FUNCTION_BLOCK "PIDControl"
{ S7_Optimized_Access := 'TRUE' }
VERSION : 0.1
AUTHOR : 'AI_Generated'

VAR_INPUT
    bEnable : Bool;                    // PID 使能
    bReset : Bool;                     // 积分复位
    bManualMode : Bool;                // 手动模式
    rSetpoint : Real;                  // 设定值 (工程单位)
    rProcessValue : Real;              // 过程值 (工程单位)
    rManualValue : Real;               // 手动输出值 (%)
    rKp : Real;                        // 比例增益
    rTi : Real;                        // 积分时间 (秒，0=无积分)
    rTd : Real;                        // 微分时间 (秒，0=无微分)
    rOutputMin : Real;                 // 输出下限 (%)
    rOutputMax : Real;                 // 输出上限 (%)
    rSetpointRampRate : Real;          // 设定值斜坡速率 (单位/秒)
    rDeadband : Real;                  // 死区 (工程单位)
END_VAR

VAR_OUTPUT
    rControlOutput : Real;             // 控制输出 (%)
    rError : Real;                     // 偏差值
    rP : Real;                         // P 分量
    rI : Real;                         // I 分量
    rD : Real;                         // D 分量
    bLimiting : Bool;                  // 输出限幅中
    bAntiWindupActive : Bool;          // 抗饱和激活
    bRampActive : Bool;                // 斜坡进行中
    rSetpointRamped : Real;            // 斜坡后的设定值
END_VAR

VAR
    // PID 内部变量
    rIntegral : Real;                  // 积分累加值
    rIntegralInc : Real;               // 本次积分增量（只计算一次）
    rPrevError : Real;                 // 上次偏差
    rPrevPV : Real;                    // 上次过程值（用于微分）
    rSampleTime : Real;                // 采样时间 (秒)
    rOutput : Real;                    // 计算输出

    // 设定值斜坡
    rRampTarget : Real;                // 斜坡目标值
    rRampCurrent : Real;               // 斜坡当前值

    // 采样周期
    tCycle : TON;                      // 采样周期定时器
    tRamp : TON;                       // 斜坡更新定时器

    // 限幅中间变量
    bOutHigh : Bool;                   // 输出超上限
    bOutLow : Bool;                    // 输出低于下限

    // 无扰切换
    bPrevManualMode : Bool;            // 上次手动模式状态
END_VAR

BEGIN
    // ── 采样周期 (200ms) ──
    // 自复位定时器：每 200ms 产生一周期脉冲，PID 计算仅在脉冲周期执行一次，
    // 而非使能后每个扫描周期都执行；rSampleTime 为采样周期对应秒数，
    // 用于斜坡步长、积分增量与微分项的时间换算
    tCycle(IN := bEnable AND NOT tCycle.Q, PT := T#200MS);
    rSampleTime := 0.2;

    IF tCycle.Q AND bEnable THEN
        // ── 设定值斜坡 ──
        IF rSetpoint <> rRampTarget THEN
            rRampTarget := rSetpoint;
            bRampActive := TRUE;
        END_IF;

        IF rSetpointRampRate > 0.0 AND rRampCurrent <> rRampTarget THEN
            IF rRampTarget > rRampCurrent THEN
                rRampCurrent := rRampCurrent + rSetpointRampRate * rSampleTime;
                IF rRampCurrent >= rRampTarget THEN
                    rRampCurrent := rRampTarget;
                    bRampActive := FALSE;
                END_IF;
            ELSE
                rRampCurrent := rRampCurrent - rSetpointRampRate * rSampleTime;
                IF rRampCurrent <= rRampTarget THEN
                    rRampCurrent := rRampTarget;
                    bRampActive := FALSE;
                END_IF;
            END_IF;
        ELSIF rSetpointRampRate <= 0.0 THEN
            // 无斜坡时直接到位
            rRampCurrent := rRampTarget;
            bRampActive := FALSE;
        END_IF;

        rSetpointRamped := rRampCurrent;

        // ── 偏差计算 ──
        rError := rSetpointRamped - rProcessValue;

        // ── 死区处理 ──
        IF ABS(rError) < rDeadband THEN
            rError := 0.0;
        END_IF;

        // ── P 分量 ──
        rP := rKp * rError;

        // ── D 分量（微分先行：对 PV 微分，避免阶跃冲击） ──
        IF rTd > 0.0 THEN
            rD := rKp * rTd * (rPrevPV - rProcessValue) / rSampleTime;
        ELSE
            rD := 0.0;
        END_IF;

        // ── I 分量（积分分离 + 抗饱和） ──
        bAntiWindupActive := FALSE;
        IF rTi > 0.0 THEN
            // 积分增量只计算一次（原实现同一周期重复两次 Real 除法）
            rIntegralInc := rKp * rError * rSampleTime / rTi;

            // 抗饱和：按当前周期预计输出（P + 当前积分 + D）判定，不再使用
            // 上一周期陈旧 rOutput；输出越限且偏差方向加剧饱和时反向积分，
            // 否则正常积分——二者互斥，避免原实现“先加后减、净效果为零”
            IF (rP + rIntegral + rD >= rOutputMax AND rError > 0.0) OR
               (rP + rIntegral + rD <= rOutputMin AND rError < 0.0) THEN
                rIntegral := rIntegral - rIntegralInc;
                bAntiWindupActive := TRUE;
            ELSIF ABS(rError) < 100.0 THEN
                // 积分分离：|偏差| > 100 时停止积分
                rIntegral := rIntegral + rIntegralInc;
            END_IF;
        END_IF;

        rI := rIntegral;

        // ── 合成输出 ──
        rOutput := rP + rI + rD;

        // ── 输出限幅 ──
        bOutHigh := FALSE; bOutLow := FALSE;
        IF rOutput > rOutputMax THEN
            rOutput := rOutputMax;
            bOutHigh := TRUE;
        ELSIF rOutput < rOutputMin THEN
            rOutput := rOutputMin;
            bOutLow := TRUE;
        END_IF;

        bLimiting := bOutHigh OR bOutLow;

        // ── 手动/自动切换（无扰切换） ──
        IF bPrevManualMode AND NOT bManualMode THEN
            // 手动→自动：初始化积分使输出无跳变
            rIntegral := rManualValue - rP - rD;
            rI := rIntegral;
            rPrevPV := rProcessValue;
            rPrevError := rError;
        END_IF;
        bPrevManualMode := bManualMode;

        IF NOT bManualMode THEN
            rControlOutput := rOutput;
        ELSE
            rControlOutput := rManualValue;
            // 自动→手动：跟踪输出，为下次切换准备
            rIntegral := rManualValue - rP - rD;
            rI := rIntegral;
        END_IF;

        // ── 更新历史值 ──
        rPrevError := rError;
        rPrevPV := rProcessValue;
    END_IF;

    // ── 复位 ──
    IF bReset THEN
        rIntegral := 0.0;
        rPrevError := 0.0;
        rPrevPV := 0.0;
        rControlOutput := 0.0;
        rRampCurrent := 0.0;
        rRampTarget := 0.0;
    END_IF;

END_FUNCTION_BLOCK
